// TIA Portal V18 export
// export: Created 2026-01-09T11:23:32.1560779Z, ExportSetting WithDefaults, DisplayName Totally Integrated Automation Portal, DisplayVersion V18 Update 5, DisplayName TIA Portal Openness, DisplayVersion V18 Update 5, DisplayName TIA Portal Teamcenter Gateway, DisplayVersion V18, DisplayName TIA Portal Version Control Interface, DisplayVersion V18, DisplayName SINAMICS Startdrive Advanced, DisplayVersion V18 SP2 Update 1, DisplayName SINAMICS Startdrive G110M, G120, G120C, G120D, G120P, G115D, DisplayVersion V18 SP2 Update 1, DisplayName SINAMICS Startdrive G130, G150, S120, S150, SINAMICS MV, S210, G220, S200, DisplayVersion V18 SP2 Update 1, DisplayName STEP 7 Professional, DisplayVersion V18 Update 5, DisplayName STEP 7 Safety, DisplayVersion V18, DisplayName WinCC Professional, DisplayVersion V18 Update 5
Screen "226_Cylinder_B2"  1280x800, Number=226, Template=02ManualUnit1
  ScreenLayer "Layer_0"
    FaceplateInstance "Cylinder_S71500_TP700_1" at 0,85 size 1279x80  FaceplateTypeName=03 FunctionBlocks@$@101 Cylinder@$@101.2 HMI@$@S7-1500@$@Cylinder_S71500_TP700 V 0.0.29
      Cy := STxxxCylinder007
      CylinderName := Cyl name
      HomeButtonName := Cyl go home button
      WorkButtonName := Cyl go work button
      HomeQaddress := Cyl home Q
      HomeIaddress := Cyl home I
      WorkIaddress := Cyl work I
      WorkQaddress := Cyl work Q
    FaceplateInstance "Cylinder_S71500_TP700_3" at 0,160 size 1279x80  FaceplateTypeName=03 FunctionBlocks@$@101 Cylinder@$@101.2 HMI@$@S7-1500@$@Cylinder_S71500_TP700 V 0.0.29
      Cy := STxxxCylinder008
      CylinderName := Cyl name
      HomeButtonName := Cyl go home button
      WorkButtonName := Cyl go work button
      HomeQaddress := Cyl home Q
      HomeIaddress := Cyl home I
      WorkIaddress := Cyl work I
      WorkQaddress := Cyl work Q
    Button "btnMenu4" at 384,725 size 128x75  Mode=Text, TextOff="读码器_806A1 / Code reader 806A1", TextOn="读码器_806A1 / Code reader 806A1"
      on Click: ActivateScreen(Screen name := 222 Scanner_806A1, Object number := 0)
    Button "btnMenu5" at 512,725 size 128x75  Mode=Text, TextOff="气缸_B2 / Cylinder _B2", TextOn="气缸_B2 / Cylinder _B2"
      on Click: ActivateScreen(Screen name := , Object number := 0)
    Button "btnMenu6" at 640,725 size 128x75  Mode=Text, TextOff="压机_375A1 / Press_375A1", TextOn="压机_375A1 / Press_375A1"
      on Click: ActivateScreen(Screen name := 227 Kistler_375A1, Object number := 0)
    Button "btnMenu6_1" at 768,725 size 128x75  Mode=Text
    Button "按钮_1" at 128,725 size 128x75  Mode=Text, PictureOff=向右箭头_0, TextOff="气缸_B1 / Cylinder _B1", TextOn="气缸_B1 / Cylinder _B1"
      on Click: ActivateScreen(Screen name := 220_Cylinder_B1, Object number := 0)
    Button "btnMenu4_1" at 256,725 size 128x75  Mode=Text, TextOff="压机_372A1 / Press_372A1", TextOn="压机_372A1 / Press_372A1"
      on Click: ActivateScreen(Screen name := 221 Kistler__372A1, Object number := 0)
    GraphicView "图形视图_1" at 284,244 size 462x443  Picture=图形_50
    Button "btnMenu7" at 896,725 size 128x75  Mode=Text
    Button "btnMenu7_1" at 1024,725 size 128x75  Mode=Text
